FUNCTION_BLOCK STACK_INTE (* A variable-size stack of INTs (with ECC) *)
  (* Standard: 61499-2 *)
  (* Version 0.0, 2004-06-07, JHC, HUT, Adapted from STACK_INT. *)
  (* Compiler header: package fb.rt.student; *)
  (* Compiler Java IBM Jikes 1.06 *)
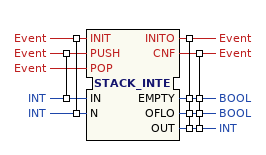
  EVENT_INPUT
    INIT WITH N; (* Empty the stack and set its maximum size to N. *)
    PUSH WITH IN; (* Push the value of IN to the top of the stack if possible. *)
    POP; (* Pop the top value off of the stack if possible. *)
  END_EVENT
  EVENT_OUTPUT
    INITO WITH EMPTY, OFLO, OUT; (* Initialization confirmation. *)
    CNF WITH EMPTY, OFLO, OUT; (* PUSH or POP confirmation. *)
  END_EVENT
  VAR_INPUT
    IN : INT; (* Input to be pushed *)
    N : INT; (* Maximum depth after INIT, 0 to 128 elements *)
  END_VAR
  VAR_OUTPUT
    EMPTY : BOOL := 1; (* Stack empty *)
    OFLO : BOOL := 0; (* Stack overflow *)
    OUT : INT := 0; (* Top of stack data (meaningless if EMPTY or OFLO). *)
  END_VAR
  VAR
    STK : ARRAY [0..127] OF INT; (* Internal stack *)
    NI : INT := 128; (* Storage for N upon reset *)
    PTR : INT := -1; (* Stack pointer *)
  END_VAR
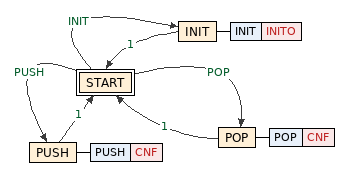
  EC_STATES
    START; (* Initial State *)
    INIT : INIT -> INITO;
    POP : POP -> CNF;
    PUSH : PUSH -> CNF;
  END_STATES
  EC_TRANSITIONS
    START TO INIT := INIT;
    INIT TO START := 1;
    START TO POP := POP;
    POP TO START := 1;
    START TO PUSH := PUSH;
    PUSH TO START := 1;
  END_TRANSITIONS
  ALGORITHM INIT IN ST:
OFLO:=FALSE;EMPTY:=TRUE;PTR:=-1;
IF N<0 THEN NI:=0;
ELSIF N>127 THEN NI:=127;
ELSE NI:=N;
END_IF;
OUT:=0;
  END_ALGORITHM
  ALGORITHM POP IN ST:
IF NOT EMPTY THEN
OFLO:=FALSE;PTR:=PTR-1;EMPTY:=PTR<0;
END_IF;
IF EMPTY THEN OUT:=0;
ELSE OUT:=STK[PTR];
END_IF;
  END_ALGORITHM
  ALGORITHM PUSH IN ST:
IF NOT OFLO THEN
  EMPTY:=FALSE;PTR:=PTR+1;OFLO:=(PTR=NI);
END_IF;
IF NOT OFLO THEN OUT:=IN;STK[PTR]:=IN;
ELSE OUT:=0;
END_IF;
  END_ALGORITHM
END_FUNCTION_BLOCK
